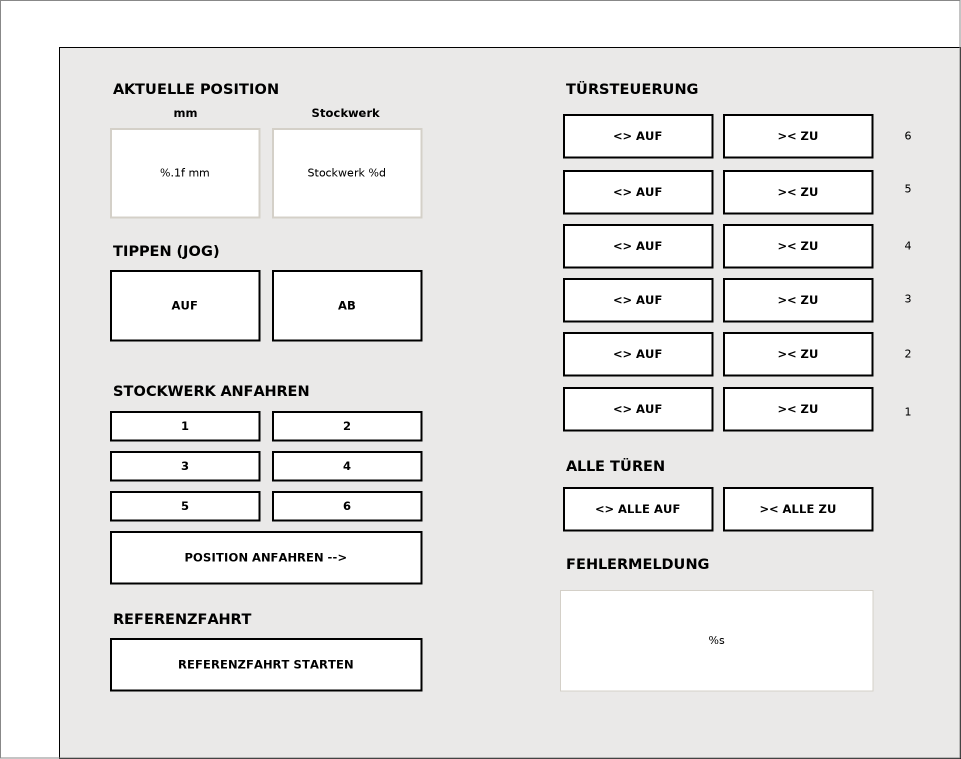
VISUALIZATION Handbetrieb  // 961x759
    RoundedRectangle (59,47 902x712)
    Textfield (110,128 150x90), "%.1f mm", text variable: Divers.AktuellePosmm
    Label (110,74 205x30), "AKTUELLE POSITION"
    Label (110,236 150x30), "TIPPEN (JOG)"
    RoundedRectangle (110,270 150x71), "AUF", colour toggle: Visu_Manuellmodus.JogAuf
        tap Visu_Manuellmodus.JogAuf
    RoundedRectangle (272,270 150x71), "AB", colour toggle: Visu_Manuellmodus.JogAb
        tap Visu_Manuellmodus.JogAb
    Label (110,376 216x30), "STOCKWERK ANFAHREN"
    RoundedRectangle (110,411 150x30), "1", colour variable: Visu_Manuellmodus.adwFloorBtnColor[1]
        OnMouseDown: execute { Visu_Manuellmodus.Zielstock := 1; }
    RoundedRectangle (272,411 150x30), "2", colour variable: Visu_Manuellmodus.adwFloorBtnColor[2]
        OnMouseDown: execute { Visu_Manuellmodus.Zielstock := 2; }
    RoundedRectangle (110,451 150x30), "3", colour variable: Visu_Manuellmodus.adwFloorBtnColor[3]
        OnMouseDown: execute { Visu_Manuellmodus.Zielstock := 3; }
    RoundedRectangle (272,451 150x30), "4", colour variable: Visu_Manuellmodus.adwFloorBtnColor[4]
        OnMouseDown: execute { Visu_Manuellmodus.Zielstock := 4; }
    RoundedRectangle (110,491 150x30), "5", colour variable: Visu_Manuellmodus.adwFloorBtnColor[5]
        OnMouseDown: execute { Visu_Manuellmodus.Zielstock := 5; }
    RoundedRectangle (272,491 150x30), "6", colour variable: Visu_Manuellmodus.adwFloorBtnColor[6]
        OnMouseDown: execute { Visu_Manuellmodus.Zielstock := 6; }
    RoundedRectangle (110,531 312x53), "POSITION ANFAHREN -->"
        tap Visu_Manuellmodus.PosAnfahren
    RoundedRectangle (110,638 312x53), "REFERENZFAHRT STARTEN"
    Label (110,604 150x30), "REFERENZFAHRT"
    Label (563,74 150x30), "TÜRSTEUERUNG"
    RoundedRectangle (563,114 150x44), "<> AUF", colour toggle: Visu_Manuellmodus.bTuerAuf[6]
        tap Visu_Manuellmodus.bTuerAuf[6]
    RoundedRectangle (723,114 150x44), ">< ZU", colour toggle: Visu_Manuellmodus.bTuerZu[6]
        tap Visu_Manuellmodus.bTuerZu[6]
    Label (883,121 50x30), "6"
    Label (883,174 50x30), "5"
    Label (883,231 50x30), "4"
    Label (883,284 50x30), "3"
    Label (883,339 50x30), "2"
    Label (883,397 50x30), "1"
    Label (563,451 150x30), "ALLE TÜREN"
    RoundedRectangle (563,487 150x44), "<> ALLE AUF"
        tap Visu_Manuellmodus.AlleTuerenAuf
    Label (83,98 205x30), "mm"
    Textfield (272,128 150x90), "Stockwerk %d", text variable: Divers.AktuellesStockwerk
    Label (243,98 205x30), "Stockwerk"
    RoundedRectangle (723,487 150x44), ">< ALLE ZU"
        tap Visu_Manuellmodus.AlleTuerenZu
    RoundedRectangle (563,170 150x44), "<> AUF", colour toggle: Visu_Manuellmodus.bTuerAuf[5]
        tap Visu_Manuellmodus.bTuerAuf[5]
    RoundedRectangle (563,224 150x44), "<> AUF", colour toggle: Visu_Manuellmodus.bTuerAuf[4]
        tap Visu_Manuellmodus.bTuerAuf[4]
    RoundedRectangle (563,278 150x44), "<> AUF", colour toggle: Visu_Manuellmodus.bTuerAuf[3]
        tap Visu_Manuellmodus.bTuerAuf[3]
    RoundedRectangle (563,332 150x44), "<> AUF", colour toggle: Visu_Manuellmodus.bTuerAuf[2]
        tap Visu_Manuellmodus.bTuerAuf[2]
    RoundedRectangle (563,387 150x44), "<> AUF", colour toggle: Visu_Manuellmodus.bTuerAuf[1]
        tap Visu_Manuellmodus.bTuerAuf[1]
    RoundedRectangle (723,170 150x44), ">< ZU", colour toggle: Visu_Manuellmodus.bTuerZu[5]
        tap Visu_Manuellmodus.bTuerZu[5]
    RoundedRectangle (723,224 150x44), ">< ZU", colour toggle: Visu_Manuellmodus.bTuerZu[4]
        tap Visu_Manuellmodus.bTuerZu[4]
    RoundedRectangle (723,278 150x44), ">< ZU", colour toggle: Visu_Manuellmodus.bTuerZu[3]
        tap Visu_Manuellmodus.bTuerZu[3]
    RoundedRectangle (723,332 150x44), ">< ZU", colour toggle: Visu_Manuellmodus.bTuerZu[2]
        tap Visu_Manuellmodus.bTuerZu[2]
    RoundedRectangle (723,387 150x44), ">< ZU", colour toggle: Visu_Manuellmodus.bTuerZu[1]
        tap Visu_Manuellmodus.bTuerZu[1]
    Textfield (560,590 313x101), "%s", text variable: Divers.Fehlertext
    Label (563,549 236x30), "FEHLERMELDUNG"
END_VISUALIZATION

(* stored: Version 1.1.0.1
   Visu Handbetrieb: Id {d2faeedd-8cfe-43c4-8ba3-765eabf19d3b} *)
